FUNCTION BIT_TOGGLE_B : BYTE
VAR_INPUT
	IN : BYTE;
	POS : INT;
END_VAR


(*
version 1.0 18. oct. 2008
programmer 	hugo
tested by	tobias

this function toggles a bit of a BYTE at position pos.

*)

BIT_TOGGLE_B := SHL(BYTE#1, POS) XOR IN;




(* revision history
hm	18. oct. 2008	rev 1.0
	original version


*)

END_FUNCTION

(* stored: Version 1.1.0.1, ProductVersion 3.1.4022.7
   POU BIT_TOGGLE_B: Id {8ee2d676-c423-4fef-bb56-6651aad7ea56}, SpecialFunc None *)
